ABB RobotStudio station: ABBDeburringStation_20211103-160115.rsstn

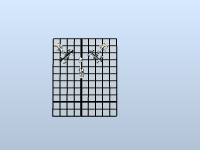
Station ABBDeburringStation (saved by RobotStudio 6.8.8307.1040)
Controller IRB6660_celdaB1, task T_ROB1: task frame (RAPID world) sits at (7800, 3200, 0) mm, rotated rx 0 ry 0 rz -140 deg in the station
Controller IRB6660_celdaA2, task T_ROB1: task frame (RAPID world) sits at (7800, -3200, 0) mm, rotated rx 0 ry 0 rz 140 deg in the station
Controller IRB6700_Master, task T_ROB1: task frame (RAPID world) sits at (4000, 0, 0) mm in the station
Controller IRB6700_Master
  mechanical unit ROB_1: IRB6700_150_320__04, 6 joints, base frame (0, 0, 0) mm
Controller IRB6660_celdaA2
  mechanical unit ROB_1: IRB6660_205_190__01, 6 joints, base frame (0, 0, 0) mm
  mechanical unit INTERCH: IRBP_R300_D1000-L1250_M2009_REV1_01, 3 joints, base frame (0, 0, 0) mm
  mechanical unit STN1: IRBP_R300_D1000-L1250_M2009_REV1_01, 1 joints, base frame (1329.58, 593.49, 950) mm, rotated rx 0 ry -90 rz 90 deg
  mechanical unit STN2: IRBP_R300_D1000-L1250_M2009_REV1_01, 1 joints, base frame (0, 0, 0) mm
Controller IRB6660_celdaB1
  mechanical unit ROB_1: IRB6660_205_190__01_2, 6 joints, base frame (0, 0, 0) mm
  mechanical unit INTERCH: IRBP_R300_D1000-L1250_M2009_REV1_01_2, 3 joints, base frame (0, 0, 0) mm
  mechanical unit STN1: IRBP_R300_D1000-L1250_M2009_REV1_01_2, 1 joints, base frame (1326.62, 649.13, 950) mm, rotated rx 0 ry -90 rz 90 deg
  mechanical unit STN2: IRBP_R300_D1000-L1250_M2009_REV1_01_2, 1 joints, base frame (0, 0, 0) mm
Layout (positions relative to the parent item):
  - IRB6700_150_320__04 [mechanism, from Robots\IRB6700_150_320__04.rslib] at (4000, 0, 0) mm; joint values [0, 0, 0, 0, 0.5236, 0] (rad or m)
  - IRB6660_205_190__01 [mechanism, from Robots\IRB6660_205_190_G_01.rslib] at (7800, -3200, 0) mm, rotated rx 0 ry 0 rz 140 deg; joint values [0, 0, 0, 0, 0.5236, 0] (rad or m)
  - IRBP_R300_D1000-L1250_M2009_REV1_01 [mechanism] at (6400, -2800, 0) mm, rotated rx 0 ry 0 rz 140 deg; joint values [0, 0, 0] (rad or m)
      links: Base, Link1, Link2, Link3
  - IRB6660_205_190__01_2 [mechanism, from Robots\IRB6660_205_190_G_01.rslib] at (7800, 3200, 0) mm, rotated rx 0 ry 0 rz -140 deg; joint values [0, 0, 0, 0, 0.5236, 0] (rad or m)
  - IRBP_R300_D1000-L1250_M2009_REV1_01_2 [mechanism] at (7201, 1850, 0) mm, rotated rx 0 ry 0 rz -140 deg; joint values [0, 0, 0] (rad or m)
      links: Base, Link1, Link2, Link3
